// TIA Portal V18 export
VAR_GLOBAL   // PLC tag table "Default tag table"
   Tag1 AT %M0.0 : Bool;
   Tag2 AT %M0.1 : Bool;
   Tag3 AT %M0.2 : Bool;
   Tag4 AT %MD10 : DInt;
   Tag5 AT %M0.4 : Bool;
   Tag6 AT %M0.5 : Bool;
   Tag7 AT %M0.6 : Bool;
   Tag8 AT %M0.7 : Bool;
   Input4 AT %I0.3 : Bool;
   Input5 AT %I0.4 : Bool;
   Input6 AT %I0.5 : Bool;
   Input7 AT %I0.6 : Bool;
   Input8 AT %I0.7 : Bool;
   Input9 AT %I1.0 : Bool;
   Input10 AT %I1.1 : Bool;
   Input11 AT %I1.2 : Bool;
   Input12 AT %I1.3 : Bool;
   Input13 AT %I1.4 : Bool;
   Input14 AT %I1.5 : Bool;
   Input15 AT %I1.6 : Bool;
   Input16 AT %I1.7 : Bool;
   Input1 AT %I0.0 : Bool;
   Input2 AT %I0.1 : Bool;
   Input3 AT %I0.2 : Bool;
   Output1 AT %Q0.0 : Bool;
   Output2 AT %Q0.1 : Bool;
   Output3 AT %Q0.2 : Bool;
   Output4 AT %Q0.3 : Bool;
   Output5 AT %Q0.4 : Bool;
   Output6 AT %Q0.5 : Bool;
   Output7 AT %Q0.6 : Bool;
   Output8 AT %Q0.7 : Bool;
   Output9 AT %Q1.0 : Bool;
   Output10 AT %Q1.1 : Bool;
   Output11 AT %Q1.2 : Bool;
   Output12 AT %Q1.3 : Bool;
   Output13 AT %Q1.4 : Bool;
   Output14 AT %Q1.5 : Bool;
   Output15 AT %Q1.6 : Bool;
   Output16 AT %Q1.7 : Bool;
   Tag_1 AT %M200.0 : Bool;
   Tag_2 AT %M200.1 : Bool;
   Tag_3 AT %M200.3 : Bool;
   Tag_4 AT %M200.4 : Bool;
   Tag_5 AT %MD410 : DWord;
   Tag_6 AT %MD420 : DWord;
   Tag_7 AT %M50.0 : Bool;
   Tag_8 AT %M50.1 : Bool;
   Tag_9 AT %M50.2 : Bool;
END_VAR
